// TIA Portal V17 export
// export: Created 2024-09-03T21:54:54.4231018Z, ExportSetting WithDefaults, DisplayName Totally Integrated Automation Portal, DisplayVersion V17 Update 7, DisplayName TIA Portal Openness, DisplayVersion V17 Update 7, DisplayName TIA Portal Version Control Interface, DisplayVersion V17, DisplayName SINAMICS Startdrive Advanced, DisplayVersion V17 SP2, DisplayName SINAMICS Startdrive G110M, G120, G120C, G120D, G120P, G115D, DisplayVersion V17 SP2, DisplayName SINAMICS Startdrive G130, G150, S120, S150, SINAMICS MV, S210, DisplayVersion V17 SP2, DisplayName STEP 7 Professional, DisplayVersion V17 Update 7, DisplayName STEP 7 Safety, DisplayVersion V17 Update 6, DisplayName WinCC Advanced / Unified PC, DisplayVersion V17 Update 7
DATA_BLOCK "DB_Main_Instance"   // DB5000
VERSION : 0.1
// stored: AutoNumber false, DBAccessibleFromOPCUA true, DBAccessibleFromWebserver true, InstanceOfName FB_Main, InstanceOfType FB
"FB_Main"
   // VAR
   //    IEC_Timer_0_Instance { S7_SetPoint := 'True'} : TON_TIME;
   //    MachineModeOld { S7_SetPoint := 'True'} : UInt := 1;
   //    F_TRIG_Instance { S7_SetPoint := 'True'} : F_TRIG;
   //    F_TRIG_Instance_1 { S7_SetPoint := 'True'} : F_TRIG;
   //    F_TRIG_Instance_2 { S7_SetPoint := 'True'} : F_TRIG;
   //    R_TRIG_Instance { S7_SetPoint := 'True'} : R_TRIG;
   //    R_TRIG_Instance_1 { S7_SetPoint := 'True'} : R_TRIG;
   // END_VAR
BEGIN
   IEC_Timer_0_Instance.PT := T#0MS;
   IEC_Timer_0_Instance.IN := FALSE;
   F_TRIG_Instance.CLK := FALSE;
   F_TRIG_Instance.Q := FALSE;
   F_TRIG_Instance.Stat_Bit := FALSE;
   F_TRIG_Instance_1.CLK := FALSE;
   F_TRIG_Instance_1.Q := FALSE;
   F_TRIG_Instance_1.Stat_Bit := FALSE;
   F_TRIG_Instance_2.CLK := FALSE;
   F_TRIG_Instance_2.Q := FALSE;
   F_TRIG_Instance_2.Stat_Bit := FALSE;
   R_TRIG_Instance.CLK := FALSE;
   R_TRIG_Instance.Q := FALSE;
   R_TRIG_Instance.Stat_Bit := FALSE;
   R_TRIG_Instance_1.CLK := FALSE;
   R_TRIG_Instance_1.Q := FALSE;
   R_TRIG_Instance_1.Stat_Bit := FALSE;
END_DATA_BLOCK
